Universal Robots PolyScope program: template_vision.urp

Program template_vision (createdIn=3.3.0.0 lastSavedIn=0.0.0.0 installation=default)
BeforeStart
  'Set gripper initial state here.'
Robot Program (runOnlyOnce=false motionType=MoveJ speed=1.047198 acceleration=1.396263 recalculateMotions=false)
  MoveJ speed 60 deg/s, acceleration 80 deg/s^2 (recalculateMotions=false)
    Waypoint Snapshot_pos: 
  URCap com.robotiq.Robotiq_Wrist_Camera.Camera Locate
    'If an object is located,'
    'these instructions are executed.'
    MoveL speed 250 mm/s, acceleration 1200 mm/s^2 (recalculateMotions=false) feature(featureName=Your_Snapshot)
      'The robot moves relatively'
      'to the located object.'
      Waypoint Rel_approach: 
      Waypoint Rel_pick: 
      'Enter your gripper instructions here.'
      Waypoint Rel_retract: 
    MoveJ speed 60 deg/s, acceleration 80 deg/s^2 (recalculateMotions=false)
      'The robot moves to absolute waypoints.'
      Waypoint Abs_approach: 
      Waypoint Abs_place: 
      'Enter your gripper instructions here.'
      Waypoint Abs_retract: 
